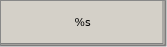
VISUALIZATION VISU_M3TargetDialogButton  // 167x47
VAR_IN_OUT
	ref : M3TargetDialogButton;
END_VAR
    Button (0,0 165x45), "%s", text variable: ref.text, input disabled if: ref.deactivate
        p2073431371: ref.fontSize
        p1845689383: ref.fontFlags
        OnMouseClick: execute { ref.do_request := TRUE; }
        OnMouseClick: CloseDialog Dialog=VISU_M3TargetDialog, Result=OK, NumpadKeypadSet=True
END_VISUALIZATION

(* stored: Version 1.1.0.1, ProductVersion 3.1.0.36
   Visu VISU_M3TargetDialogButton: Id {fade314e-6317-4ec5-a758-b16378190053} *)
